// TIA Portal V18 export
TYPE "PLCtoMES_MainCheckOutProcessData_OP220"
// stored: IsFailsafeCompliant false
   STRUCT
      "P-LineID" : String[18];   // 生产线代号
      "P-StationID" : String[18];   // 工位代号
      "P-PalletNo" : Int;   // 托盘编号
      "P-PalletType" : Byte;   // 托盘类型，1-LOOP1托盘，2-LOOP2托盘等
      "P-PalletStatus" : Byte;   // 预留 托盘状态
      "P-CT_Total" : Real;   // 总循环时间（秒），当前工件开始加工后由PLC累积加工时长，工件离开后停止累计时长
      "P-CT_Sub" : Array[1..20] of Real;   // 工步分项节拍时间（秒），比如物流时间，工步1时间，工步2时间等
      "P-Data" { S7_SetPoint := 'True'} : "PLCtoMES_OP_ProcessData_OP220";   // 质量终值数据数组
      Reserve { S7_SetPoint := 'True'} : Array[1..1700] of Byte;   // CheckOutProcessData预留
   END_STRUCT;
END_TYPE
